{attribute 'qualified_only'}
VAR_GLOBAL

	eCommand : E_Command;
END_VAR

(* stored: Version 1.1.0.1, ProductVersion 3.1.4024.11
   GVL Command: Id {461a0450-000e-4fb8-9b96-604c62830b5c} *)
